Fanuc KAREL source: kt00206.KL

PROGRAM KT00206
%STACKSIZE=65535
%PRIORITY=65535
%NOLOCKGROUP
VAR
I1 : INTEGER
Y2 : ARRAY[2] OF BYTE
OUT : INTEGER
BEGIN
I1=2
Y2[1]=3
-- UNRESOLVED_PC line 10 opcodes [21 22 9D 33 B1 46 23] marker_code=35
END KT00206
